(* CoDeSys 2.3.9.41 project: mixer.pro *)

(* Task configuration *)
TASK NewTask (PRIORITY := 1); (* freewheeling *)
	VIS_PRG();
	PLC_PRG();
END_TASK

(* Global variable list: Global_Variables *)
VAR_GLOBAL

(*Входы*)

(*Кнопки*)
	PBSTRT: BOOL; (*Кнопка налить*)
	PBStop: BOOL; (*Кнопка возврат*)

(*Датчики*)
	DU1: BOOL; (*Датчик уровня бака 1*)
	DU2: BOOL; (*Датчик уровня бака 2*)
	U0: BOOL; (*Уров. 0 в мерной емкости*)
	U1: BOOL;(*Уров. 1 в мерной емкости*)
	DB: BOOL;(*Датчик тары*)
	M: BOOL;(*Датчик монеты*)

(*Датчики компаратора*)
	PM1: BOOL;(*Принята монета 1*)
	PM2: BOOL;(*Принята монета 2*)
	PM5: BOOL;(*Принята монета 5*)
	PM10: BOOL;(*Принята монета 10*)

(*Выходы*)

(*Приводы/устройства*)
	KL0: BOOL;(*Открыть клапан 0*)
	KL1: BOOL;(*Открыть клапан 1*)
	KL2: BOOL;(*Открыть клапан 2*)
	Kk: BOOL;(*Открыть крышку камеры*)
	Zn: BOOL;(*Открыть заслонку накопителя*)
	Zsb: BOOL;(*Открыть заслонку сброса*)
	Zs: BOOL;(*Открыть заслонку сейфа*)
	Zv: BOOL;(*Открыть заслонку выдачи*)
	Com: BOOL;(*Включить компаратор*)

(*Состояния/лампы*)
	RT: BOOL; (*Состаяние возврата монет*)
	SysOn: BOOL; (*Состояние разлива*)
	FE1: BOOL;(*Фляга 1 пуста*)
	FE2: BOOL;(*Фляга 2 пуста*)
	TE: BOOL;(*Отсутствует тара*)
	Vref: BOOL;(*Режим возврата монет*)
	Nn: BOOL;(*Напиток наливается*)
	Nn1: BOOL; (*Состояние разлива 1 напитка*)
	Nn2: BOOL; (*Состояние разлива 2 напитка*)

(*Дисплей*)
	Num1_1: BOOL;(*Первая цифра старшего разряда суммы*)
	Num1_2: BOOL;(*Вторая цифра старшего разряда суммы*)
	Num2_1: BOOL;(*Первая цифра младшего разряда суммы*)
	Num2_2: BOOL;(*Вторая цифра младшего разряда суммы*)
	Num2_3: BOOL;(*Третья цифра младшего разряда суммы*)
	Num2_4: BOOL;(*Четвертая цифра младшего разряда суммы*)

	Sum15: BOOL; (*Сумма монет в монетоприемнике равна 15*)
	Sum25: BOOL; (*Сумма монет в монетоприемнике равна 25*)

END_VAR

(* POU VIS_PRG, ST *)
PROGRAM VIS_PRG
VAR
	PBTnk1: BOOL;
	PBCmp1: BOOL;
	Cmp1, _Cmp1: INT;              (* объем компонента 1 (синего)   в баке 1 *)
	PBTnk2: BOOL;
	PBCmp2: BOOL;
	Cmp2, _Cmp2: INT;              (* объем компонента 2 (красного)   в баке 2 *)
	Cmp3, _Cmp3: INT;
	ClrCmp3: DWORD;
	Mix: INT;
	_Mix: INT;
	MixClr: DWORD;
	Color: INT;
	Coin1, _Coin1: INT;
	Coin2, _Coin2: INT;
	Coin5, _Coin5: INT;
	Coin10, _Coin10: INT;
	Coin0, _Coin0:  INT;
	inputShift, _inputShift: INT;
	NUM1: INT;
	NUM2: INT;
	NUM3,  _NUM3: INT;
	PBCoin1: BOOL;
	PBCoin2: BOOL;
	PBCoin5: BOOL;
	PBCoin10: BOOL;
	PBCoin0: BOOL;
	CoinMovement: BOOL;
	CoverShift, _CoverShift: INT;
	StorageShift, _StorageShift: INT;
	SafeShift, _SafeShift: INT;
	Count1, Count2, Count5, Count10: INT;
	SUM1: INT; (*Сумма в накопителе*)

END_VAR
(*Рассчет объема компонент в каждом из баков*)
Cmp1:= MAX(0,MIN(300,BOOL_TO_INT(NOT PBCmp1)*_Cmp1+BOOL_TO_INT(PBTnk1)*300-BOOL_TO_INT(KL1)));
Cmp2:= MAX(0,MIN(300,BOOL_TO_INT(NOT PBCmp2)*_Cmp2+BOOL_TO_INT(PBTnk2)*300-BOOL_TO_INT(KL2)));

DU1:=(Cmp1>0);               (* датчик нулевого уровня бака 1*)
DU2:=(Cmp2>0);               (* датчик нулевого уровня бака 2 *)

Mix:=MAX(0,MAX(0,MIN(60, _Mix+BOOL_TO_INT(KL1)*2 + BOOL_TO_INT(KL2 )*2-BOOL_TO_INT(KL0))));
Color := MAX(BOOL_TO_INT(Nn1), 1 - BOOL_TO_INT(Nn2));

Cmp3:=MAX(0,MIN(60, _Cmp3+BOOL_TO_INT(KL0)));

MixClr := 65536*REAL_TO_BYTE(255*Color)+REAL_TO_BYTE(255*(1-Color));
ClrCmp3:=MixClr;

IF NOT M AND (PBCoin1 OR PBCoin2 OR PBCoin5 OR PBCoin10 OR PBCoin0) THEN CoinMovement:= 1;
END_IF;

Coin1:=  MAX(0, MIN(230,BOOL_TO_INT(PBCoin1)+ _Coin1 + BOOL_TO_INT(CoinMovement AND (_Coin1>0))*10)) * BOOL_TO_INT(CoinMovement AND NOT(INT_TO_BOOL(_Coin2+_Coin5+_Coin10+_Coin0)));
Coin2:=  MAX(0, MIN(280,BOOL_TO_INT(PBCoin2)+ _Coin2 + BOOL_TO_INT(CoinMovement AND (_Coin2>0))*10)) * BOOL_TO_INT(CoinMovement AND NOT(INT_TO_BOOL(_Coin1+_Coin5+_Coin10+_Coin0)));
Coin5:=  MAX(0, MIN(330,BOOL_TO_INT(PBCoin5)+ _Coin5 + BOOL_TO_INT(CoinMovement AND (_Coin5>0))*10)) *  BOOL_TO_INT(CoinMovement AND NOT(INT_TO_BOOL(_Coin2+_Coin1+_Coin10+_Coin0)));
Coin10:=  MAX(0, MIN(380,BOOL_TO_INT(PBCoin10)+ _Coin10 + BOOL_TO_INT(CoinMovement AND (_Coin10>0))*10)) * BOOL_TO_INT(CoinMovement AND NOT(INT_TO_BOOL(_Coin2+_Coin5+_Coin1+_Coin0)));
Coin0:=  MAX(0, MIN(430,BOOL_TO_INT(PBCoin0)+ _Coin0 + BOOL_TO_INT(CoinMovement AND (_Coin0>0))*2)) * BOOL_TO_INT(CoinMovement AND NOT(INT_TO_BOOL(_Coin2+_Coin5+_Coin10+_Coin1)));

IF (_Coin1 = 230 OR _Coin2 = 280 OR _Coin5 = 330 OR _Coin10 = 380 OR _Coin0 = 430) AND CoinMovement THEN
M:=1;
NUM3:=  BOOL_TO_INT(INT_TO_BOOL(Coin1)) + BOOL_TO_INT(INT_TO_BOOL(Coin2)) * 2 + BOOL_TO_INT(INT_TO_BOOL(Coin5)) * 5 + BOOL_TO_INT(INT_TO_BOOL(Coin10)) * 10;
SUM1:= SUM1 + NUM3;
CoinMovement:= 0;
Coin1:=0;
Coin2:=0;
Coin5:=0;
Coin10:=0;
Coin0:=0;
END_IF;

Sum15 := (SUM1 >= 15 AND SUM1 < 25);
Sum25 := (SUM1 = 25);

CoverShift := MAX(0, MIN(80, BOOL_TO_INT(M) + _CoverShift - BOOL_TO_INT(NOT Kk) ));

PM1 := (NUM3 = 1) AND M AND (CoverShift = 80);
PM2 := (NUM3 = 2) AND M AND (CoverShift = 80);
PM5 := (NUM3 = 5) AND M AND (CoverShift = 80);
PM10 := (NUM3 = 10) AND M AND (CoverShift = 80);

StorageShift := MAX(0, MIN(60, BOOL_TO_INT(PM1 OR PM2 OR PM5 OR PM10) + _StorageShift  - BOOL_TO_INT(NOT M AND _CoverShift <= 80) ));

SafeShift := MAX(0, MIN(60, BOOL_TO_INT(SysOn)+_SafeShift - BOOL_TO_INT(NOT Zs)));

inputShift := MAX(0, MIN(60, BOOL_TO_INT(Vref) + _inputShift - BOOL_TO_INT(NOT Zv) ));

(*_NUM3:= NUM3 * BOOL_TO_INT(StorageShift = 60); *)

(*M:= (StorageShift = 60 AND CoverShift = 80) OR NOT (StorageShift = 0 AND CoverShift = 0);*)
(*M:= (StorageShift = 60 AND CoverShift = 80) ;*)

(*NUM1 := BOOL_TO_INT(Num1_1)  * 2 + BOOL_TO_INT(Num1_2) * 1;
NUM2 := BOOL_TO_INT(Num2_1) * 8 + BOOL_TO_INT(Num2_2) * 4 + BOOL_TO_INT(Num2_3) * 2 + BOOL_TO_INT(Num2_4) * 1;*)

U0 := (Mix>0);
U1 := (Mix>=60);

IF ( StorageShift = 60) THEN
NUM2:= SUM1 MOD 10;
NUM1:= SUM1 / 10;
M:=0;
END_IF

IF (StorageShift = 60 AND M = 0) THEN
Count1:= Count1 +  BOOL_TO_INT(PM1);
Count2:= Count2 +  BOOL_TO_INT(PM2);
Count5:= Count5 +  BOOL_TO_INT(PM5);
Count10:= Count10 +  BOOL_TO_INT(PM10);
NUM3:=0;
(*StorageShift:=0;*)
(*CoverShift:=0;*)
END_IF

_Cmp1:=Cmp1;
_Cmp2:=Cmp2;
_Cmp3:=Cmp3;
_Mix:=Mix;
_Coin1:=Coin1;
_Coin2:=Coin2;
_Coin5:=Coin5;
_Coin10:=Coin10;
_Coin0:=Coin0;
_CoverShift := CoverShift;
_StorageShift := StorageShift;
_SafeShift := SafeShift;
_NUM3:= NUM3;
_inputShift := inputShift;
END_PROGRAM

(* POU PLC_PRG, ST *)
PROGRAM PLC_PRG
VAR
	_SysOn: BOOL;
	_Nn: BOOL;
	_Vref: BOOL;
	_RT: BOOL;
	_Nn1: BOOL;
	_Nn2: BOOL;
	_KL0, _KL1, _KL2: BOOL;
	Nm, _Nm: BOOL; (*Состояние разлива в мерную емкость*)
END_VAR
(*7. Переход в и из состояния возврата монет*)
IF NOT _SysOn AND PBStop THEN Vref := 1;
ELSIF NOT PBStop AND _Vref THEN Vref := 0;
END_IF;

(*8. Переходы в и из состояния разлива напитков*)
IF NOT _SysOn AND PBSTRT AND (Sum15 OR Sum25 ) THEN SysOn:=1;                              (* SysOn+  *)
ELSIF  _SysOn  AND PBStop OR ( KL0 AND NOT (U0 OR U1)) THEN SysOn:=0;                           (* SysOn-  *)
END_IF;

IF _SysOn AND DU1 AND NOT Vref AND Sum15 AND NOT _Nn1 THEN Nn1:=1;
ELSIF (NOT _SysOn OR NOT DU1 OR Vref OR NOT Sum15) AND _Nn1 THEN Nn1:=0;
END_IF;

IF _SysOn AND DU2 AND NOT Vref AND Sum25 AND NOT _Nn2 THEN Nn2:=1;
ELSIF (NOT _SysOn OR NOT DU2 OR Vref OR NOT Sum25) AND _Nn2 THEN Nn2:=0;
END_IF;

IF Nn1 AND NOT U1 AND NOT KL0 AND NOT _KL1 AND NOT _KL2  AND _SysOn THEN KL1 := 1;
ELSIF Nn1 AND U1 AND KL0 AND _KL1  THEN KL1:=0;
END_IF;

IF Nn2 AND NOT U1 AND NOT KL0 AND NOT _KL2 AND NOT _KL1 AND _SysOn THEN KL2 := 1;
ELSIF Nn2 AND U1 AND KL0 AND _KL2 THEN KL2:=0;
END_IF;

(*KL1 := Nn1 AND NOT U1;
KL2 := Nn2 AND NOT U1 AND NOT KL0;*)

IF (Nn1 OR Nn2) AND DB AND U1 AND NOT _KL0 AND _SysOn THEN KL0 := 1;
ELSIF (Nn1 OR Nn2) AND DB AND NOT U0 AND _KL0 THEN KL0 := 0;
END_IF;

(*11. Заслонка выдачи*)
IF NOT _SysOn AND _Vref THEN Zv := 1;
ELSIF _SysOn AND NOT _Vref THEN Zv := 0;
END_IF;

(*12. Сейфовая заслонка*)
IF NOT _Vref AND _SysOn THEN Zs := 1;
ELSIF _Vref AND NOT _SysOn THEN Zs := 0;
END_IF;

(*15. Крышка монетной камеры*)
IF NOT M AND NOT Nn AND NOT Vref THEN Kk := 0;
ELSIF M OR Nn OR Vref THEN Kk := 1;
END_IF;

DB := (Nn1 OR Nn2) OR (Sum15 OR Sum25);

(* ------- Лампы ------- *)
FE1 := NOT DU1;                                                                (* TS1Lmp  *)
FE2:= NOT DU2;                                                                (* TS2Lmp  *)
TE:= NOT DB;

_Vref := Vref;
_SysOn:=SysOn;
_Nn1:= Nn1;
_Nn2:=Nn2;
_Nm:=Nm;
_KL0 := KL0;
_KL1 := KL1;
_KL2 := KL2;
END_PROGRAM

(* Visualisation vis_mixer
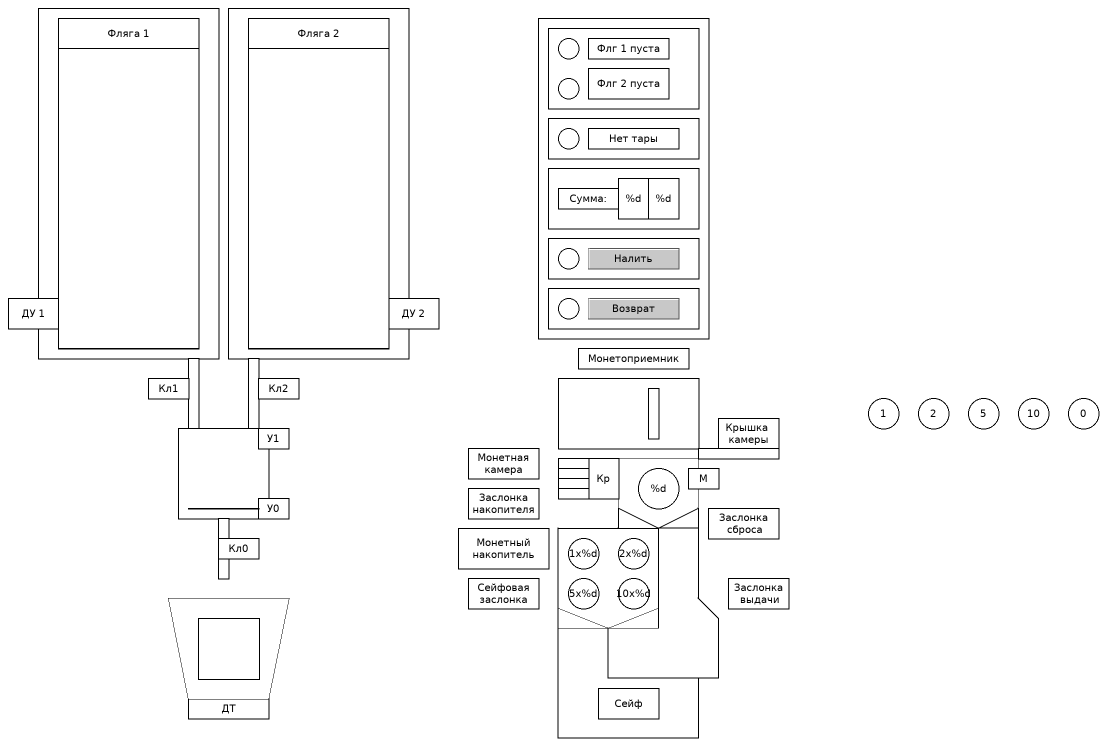
ellipse at (910,60)-(931,81): alarm colour if .FE1
ellipse at (910,100)-(931,121): alarm colour if .FE2
ellipse at (910,150)-(931,171): alarm colour if .TE
ellipse at (910,320)-(931,341): alarm colour if .Vref
ellipse at (910,270)-(931,291): alarm colour if .SysOn
button at (940,270)-(1031,291): text "Налить"; taps PBSTRT
button at (940,320)-(1031,341): text "Возврат"; taps .PBStop
rectangle at (360,320)-(411,351): text "ДУ 1"; alarm colour if DU1
rectangle at (740,320)-(791,351): text "ДУ 2"; alarm colour if DU2
rectangle at (500,400)-(541,421): text "Кл1"; alarm colour if .KL1
rectangle at (610,400)-(651,421): text "Кл2"; alarm colour if .KL2
rectangle at (610,450)-(641,471): text "У1"; alarm colour if U1
rectangle at (610,520)-(641,541): text "У0"; alarm colour if U0
rectangle at (570,560)-(611,581): text "Кл0"; alarm colour if .KL0
rectangle at (540,720)-(621,741): text "ДТ"; taps .DB
rectangle at (410,40)-(551,71): text "Фляга 1"
rectangle at (600,40)-(741,71): text "Фляга 2"
rectangle at (940,60)-(1021,81): text "Флг 1 пуста"
rectangle at (940,90)-(1021,121): text "Флг 2 пуста"
rectangle at (940,150)-(1031,171): text "Нет тары"
rectangle at (410,70)-(551,371): taps VIS_PRG.PBTnk1
rectangle at (600,70)-(741,371): taps VIS_PRG.PBTnk2
rectangle at (930,370)-(1041,391): text "Монетоприемник"
ellipse at (1220,420)-(1251,451): text "1"; invisible if VIS_PRG.Coin1=230; taps .VIS_PRG.PBCoin1; x offset -.VIS_PRG.Coin1
ellipse at (1270,420)-(1301,451): text "2"; invisible if VIS_PRG.Coin2=280; taps .VIS_PRG.PBCoin2; x offset -.VIS_PRG.Coin2
ellipse at (1320,420)-(1351,451): text "5"; taps VIS_PRG.PBCoin5; x offset -.VIS_PRG.Coin5
ellipse at (1370,420)-(1401,451): text "10"; taps VIS_PRG.PBCoin10; x offset -.VIS_PRG.Coin10
rectangle at (910,210)-(971,231): text "Сумма:"
rectangle at (970,200)-(1001,241): text "%d"; shows VIS_PRG.NUM1
rectangle at (1000,200)-(1031,241): text "%d"; shows VIS_PRG.NUM2
rectangle at (1080,600)-(1141,631): text "Заслонка / выдачи"
rectangle at (1070,440)-(1131,471): text "Крышка / камеры"
rectangle at (950,710)-(1011,741): text "Сейф"
rectangle at (820,600)-(891,631): text "Сейфовая / заслонка"
rectangle at (1060,530)-(1131,561): text "Заслонка / сброса"
rectangle at (820,510)-(891,541): text "Заслонка / накопителя"
rectangle at (810,550)-(901,591): text "Монетный / накопитель"
rectangle at (820,470)-(891,501): text "Монетная / камера"
ellipse at (990,490)-(1031,531): text "%d"; shows .VIS_PRG.NUM3 * BOOL_TO_INT(M)
rectangle at (1040,490)-(1071,511): text "М"; alarm colour if .M
rectangle at (410,370)-(551,371): taps VIS_PRG.PBCmp1; bottom -VIS_PRG.Cmp1
rectangle at (600,370)-(741,371): taps VIS_PRG.PBCmp2; bottom -VIS_PRG.Cmp2
ellipse at (1420,420)-(1451,451): text "0"; taps VIS_PRG.PBCoin0; x offset -.VIS_PRG.Coin0
rectangle at (1050,470)-(1131,481): x offset -VIS_PRG.CoverShift
rectangle at (940,480)-(971,521): text "Кр"
rectangle at (910,480)-(941,491): alarm colour if .PM1
rectangle at (910,490)-(941,501): alarm colour if .PM2
rectangle at (910,500)-(941,511): alarm colour if .PM5
rectangle at (910,510)-(941,521): alarm colour if .PM10
polygon at (960,630)-(1010,650): angle -VIS_PRG.inputShift
polygon at (910,630)-(960,650): angle VIS_PRG.SafeShift
polyline at (970,530)-(1010,550): angle VIS_PRG.StorageShift
ellipse at (970,600)-(1001,631): text "10x%d"; shows VIS_PRG.Count10; taps VIS_PRG.PBCoin10
ellipse at (920,600)-(951,631): text "5x%d"; shows VIS_PRG.Count5
ellipse at (920,560)-(951,591): text "1x%d"; shows 1 * VIS_PRG.Count1; taps .VIS_PRG.PBCoin1
ellipse at (970,560)-(1001,591): text "2x%d"; shows VIS_PRG.Count2; taps .VIS_PRG.PBCoin2
22 more shapes without text or variables
2 elements of other kinds (tables, trends, ...) not read
*)
